Universal Robots PolyScope program: ad_feasure_46.urp

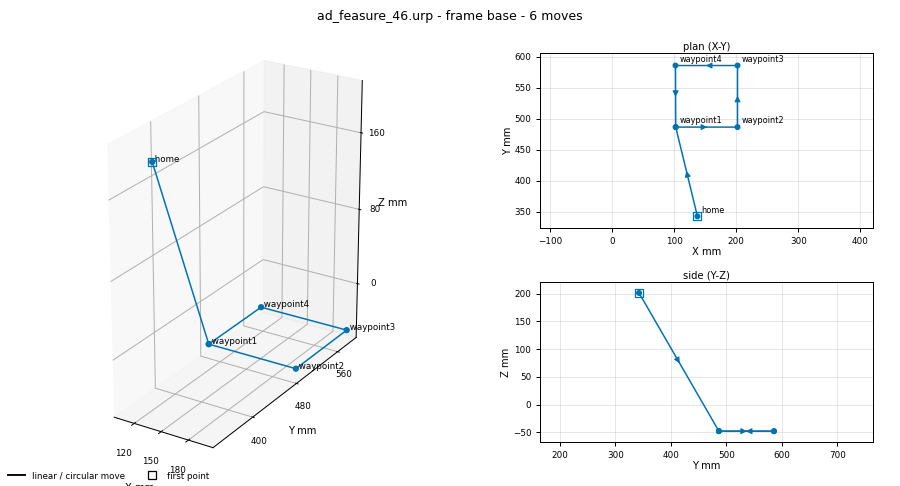
[picture p0: tool path of ad_feasure_46.urp in frame base, 6 of 6 moves have a stored position in this frame; points joined in program order, loops and branches not executed]
Program ad_feasure_46 (createdIn=3.2.19293 lastSavedIn=3.2.19293 directory=/programs installation=default robotSerialNumber=2015351391)
Calibrated DH parameters: a=[0.000352, -0.161198, -0.373486, 0.00005, 0.000049, 0]; d=[0.089268, 352.477598, -320.08558, -32.281492, 0.094939, 0.082518]; alpha=[1.570728, 0.001116, -0.003686, 1.571189, -1.570572, 0]; deltaTheta=[-0.000012, 1.181849, -1.491165, 0.309495, -0.000007, 0.000025]
Robot Program (runOnlyOnce=false motionType=MoveJ speed=1.047198 acceleration=1.396263 recalculateMotions=false)
  MoveJ speed 60 deg/s, acceleration 80 deg/s^2 (recalculateMotions=false)
    Waypoint home: TCP in base x=137.397 y=342.808 z=201.457 mm, rx=-3.1064 ry=-0.0331 rz=-0.027 rad; joints [86.157, -71.682, -121.149, -75.124, 88.93, -5.179] deg; flange x=135.274 y=338.406 z=326.321 mm, rx=-3.1065 ry=-0.0331 rz=-0.0269 rad
    MoveL speed 250 mm/s, acceleration 1200 mm/s^2 (recalculateMotions=false) feature=plane_1
      Waypoint waypoint1: TCP in base x=102.39 y=486.732 z=-47.679 mm, rx=3.1289 ry=0.1463 rz=-0.0417 rad; joints [90.411, -113.01, -121.605, -35.991, 91.397, -5.177] deg; pose in feature x=-136.879 y=164.206 z=-76.044 mm, rx=-0.0518 ry=-0.1042 rz=1.4216 rad; flange x=105.651 y=488.001 z=77.258 mm, rx=3.1289 ry=0.1463 rz=-0.0417 rad
      Waypoint waypoint2: TCP in base x=202.02 y=486.692 z=-47.702 mm, rx=3.1288 ry=0.1464 rz=-0.0416 rad; joints [79.112, -115.812, -116.577, -38.502, 91.245, -16.481] deg; pose in feature x=-131.431 y=263.685 z=-75.436 mm, rx=-0.052 ry=-0.1043 rz=1.4216 rad; flange x=205.267 y=488.002 z=77.245 mm, rx=3.1288 ry=0.1464 rz=-0.0416 rad
      Waypoint waypoint3: TCP in base x=202.048 y=585.981 z=-47.729 mm, rx=3.1287 ry=0.1464 rz=-0.0416 rad; joints [80.868, -124.675, -100.391, -45.79, 91.256, -14.72] deg; pose in feature x=-32.714 y=258.211 z=-66.318 mm, rx=-0.052 ry=-0.1043 rz=1.4216 rad; flange x=205.285 y=587.303 z=77.224 mm, rx=3.1287 ry=0.1464 rz=-0.0417 rad
      Waypoint waypoint4: TCP in base x=102 y=585.986 z=-47.759 mm, rx=3.1286 ry=0.1466 rz=-0.0416 rad; joints [90.392, -122.207, -105.078, -43.335, 91.374, -5.2] deg; pose in feature x=-47.563 y=158.285 z=33.373 mm, rx=-0.0553 ry=-0.1069 rz=1.4211 rad; flange x=105.26 y=587.278 z=77.196 mm, rx=3.1286 ry=0.1465 rz=-0.0416 rad
      Waypoint waypoint1: TCP in base x=102.39 y=486.732 z=-47.679 mm, rx=3.1289 ry=0.1463 rz=-0.0417 rad; joints [90.411, -113.01, -121.605, -35.991, 91.397, -5.177] deg; pose in feature x=-136.879 y=164.206 z=-76.044 mm, rx=-0.0518 ry=-0.1042 rz=1.4216 rad; flange x=105.651 y=488.001 z=77.258 mm, rx=3.1289 ry=0.1463 rz=-0.0417 rad
